FUNCTION_BLOCK POU_XaxisCtrl
VAR_INPUT
END_VAR
VAR_OUTPUT
END_VAR
VAR
END_VAR

// NETWORK 1

END_FUNCTION_BLOCK

(* stored: Version 1.1.0.1, ProductVersion 3.1.4024.2
   POU POU_XaxisCtrl: Id {e16decf4-0fcd-4a60-930a-cff38417a2d7}, SpecialFunc None *)
